// TIA Portal V21 export
VAR_GLOBAL   // PLC tag table "K_Analogica_Filler"
END_VAR
VAR_GLOBAL CONSTANT   // user constants
   K_Analogica_Filler_TemperaturaSalamoia : Int := 0;
   K_Analogica_Filler_TemperaturaOlio : Int := 0;
   K_Analogica_Filler_ProductTankLevel : Int := 0;
   K_Analogica_Filler_TemperaturaProdVasca : Int := 0;
   K_Analogica_Filler_TemperaturaProdIngresso : Int := 0;
   K_Analogica_Filler_LivelloSerbatoioVuoto : Int := 0;
END_VAR
